(* IEC 61131-3 sources: volt/packages/volt-lsp-iec/test-corpus/awa-palletizer/Device/Plc Logic/Application/Library Manager/IoStandard, 21 files *)

(* ---- SVN_INFO_FLAGS.gvl ---- *)
VAR_GLOBAL
	XINCOMPLETE : BOOL := FALSE;
	XMODIFIED : BOOL := TRUE;
	XSWITCHED : BOOL := FALSE;
	XCLEAN : BOOL := FALSE;
	XDISCONNECTED : BOOL := FALSE;
END_VAR

(* ---- SVN_INFO_LASTCHANGE.gvl ---- *)
VAR_GLOBAL
	DTLASTCHANGEUTC : DATE_AND_TIME := DATE_AND_TIME#2021-2-4-15:22:35;
	WSLASTCHANGELOCAL : WSTRING(44) := "2021-02-04 16:22:35 +0100 (Thu, 04 Feb 2021)";
	WSLASTCHANGEAUTHOR : WSTRING(8) := "b.schurr";
END_VAR

(* ---- SVN_INFO_REVISIONS.gvl ---- *)
VAR_GLOBAL
	LIMINREVISION : LINT := LINT#52494;
	LIMAXREVISION : LINT := LINT#52494;
END_VAR

(* ---- SVN_INFO_SUMMARY.gvl ---- *)
VAR_GLOBAL
	SVERSIONSUMMARY : STRING(6) := '52494M';
END_VAR

(* ---- SVN_INFO_SUMMARYW.gvl ---- *)
VAR_GLOBAL
	WSVERSIONSUMMARY : WSTRING(6) := "52494M";
END_VAR

(* ---- SVN_INFO_URI.gvl ---- *)
VAR_GLOBAL
	WURL : WSTRING(94) := "svn://server04/LibrariesV3Source/branches/V3.5.17.0/Intern/IoDriverBase/IoStandard/IoStandard/";
END_VAR

(* ---- CONFIGGETCONNECTOR.pou ---- *)
FUNCTION CONFIGGETCONNECTOR : POINTER TO IoConfigConnector
VAR_INPUT
	PIOCONNECTORLIST : POINTER TO IoConfigConnector;
	PNCOUNT : POINTER TO DINT;
	DWMODULETYPE : DWORD;
	DWINSTANCE : DWORD;
END_VAR
END_FUNCTION

(* ---- CONFIGGETFIRSTCHILD.pou ---- *)
FUNCTION CONFIGGETFIRSTCHILD : POINTER TO IoConfigConnector
VAR_INPUT
	PIOCONNECTORLIST : POINTER TO IoConfigConnector;
	PNCOUNT : POINTER TO DINT;
	PFATHER : POINTER TO IoConfigConnector;
END_VAR
END_FUNCTION

(* ---- CONFIGGETFIRSTCONNECTOR.pou ---- *)
FUNCTION CONFIGGETFIRSTCONNECTOR : POINTER TO IoConfigConnector
VAR_INPUT
	PIOCONNECTORLIST : POINTER TO IoConfigConnector;
	PNCOUNT : POINTER TO DINT;
	WTYPE : WORD;
END_VAR
END_FUNCTION

(* ---- CONFIGGETNEXTCHILD.pou ---- *)
FUNCTION CONFIGGETNEXTCHILD : POINTER TO IoConfigConnector
VAR_INPUT
	PIOCONNECTORLIST : POINTER TO IoConfigConnector;
	PNCOUNT : POINTER TO DINT;
	PFATHER : POINTER TO IoConfigConnector;
END_VAR
END_FUNCTION

(* ---- CONFIGGETNEXTCONNECTOR.pou ---- *)
FUNCTION CONFIGGETNEXTCONNECTOR : POINTER TO IoConfigConnector
VAR_INPUT
	PIOCONNECTORLIST : POINTER TO IoConfigConnector;
	PNCOUNT : POINTER TO DINT;
	WTYPE : WORD;
END_VAR
END_FUNCTION

(* ---- CONFIGGETPARAMETER.pou ---- *)
FUNCTION CONFIGGETPARAMETER : POINTER TO IoConfigParameter
VAR_INPUT
	PIOCONNECTOR : POINTER TO IoConfigConnector;
	DWPARAMETERID : DWORD;
END_VAR
END_FUNCTION

(* ---- CONFIGGETPARAMETERLENGTH.pou ---- *)
FUNCTION CONFIGGETPARAMETERLENGTH : DWORD
VAR_INPUT
	PPARAMETER : POINTER TO IoConfigParameter;
END_VAR
END_FUNCTION

(* ---- CONFIGGETPARAMETERVALUEBYTE.pou ---- *)
FUNCTION CONFIGGETPARAMETERVALUEBYTE : BYTE
VAR_INPUT
	PPARAMETER : POINTER TO IoConfigParameter;
	PRESULT : POINTER TO UDINT;
END_VAR
END_FUNCTION

(* ---- CONFIGGETPARAMETERVALUEBYTE_INTERNAL.pou ---- *)
FUNCTION CONFIGGETPARAMETERVALUEBYTE_INTERNAL : BYTE
VAR_INPUT
	PPARAMETER : POINTER TO IoConfigParameter;
	PRESULT : POINTER TO UDINT;
END_VAR
END_FUNCTION

(* ---- CONFIGGETPARAMETERVALUEDWORD.pou ---- *)
FUNCTION CONFIGGETPARAMETERVALUEDWORD : DWORD
VAR_INPUT
	PPARAMETER : POINTER TO IoConfigParameter;
	PRESULT : POINTER TO UDINT;
END_VAR
END_FUNCTION

(* ---- CONFIGGETPARAMETERVALUEDWORD_INTERNAL.pou ---- *)
FUNCTION CONFIGGETPARAMETERVALUEDWORD_INTERNAL : DWORD
VAR_INPUT
	PPARAMETER : POINTER TO IoConfigParameter;
	PRESULT : POINTER TO UDINT;
END_VAR
END_FUNCTION

(* ---- CONFIGGETPARAMETERVALUEPOINTER.pou ---- *)
FUNCTION CONFIGGETPARAMETERVALUEPOINTER : POINTER TO BYTE
VAR_INPUT
	PPARAMETER : POINTER TO IoConfigParameter;
	PRESULT : POINTER TO UDINT;
END_VAR
END_FUNCTION

(* ---- CONFIGGETPARAMETERVALUEWORD.pou ---- *)
FUNCTION CONFIGGETPARAMETERVALUEWORD : WORD
VAR_INPUT
	PPARAMETER : POINTER TO IoConfigParameter;
	PRESULT : POINTER TO UDINT;
END_VAR
END_FUNCTION

(* ---- CONFIGGETPARAMETERVALUEWORD_INTERNAL.pou ---- *)
FUNCTION CONFIGGETPARAMETERVALUEWORD_INTERNAL : WORD
VAR_INPUT
	PPARAMETER : POINTER TO IoConfigParameter;
	PRESULT : POINTER TO UDINT;
END_VAR
END_FUNCTION

(* ---- PRIVATE_IOMGR_MEMCPY.pou ---- *)
FUNCTION PRIVATE_IOMGR_MEMCPY : INT
VAR_INPUT
	PSRC : POINTER TO BYTE;
	PDST : POINTER TO BYTE;
	ISIZE : INT;
END_VAR
END_FUNCTION
